FUNCTION_BLOCK FB_PostPalletizer EXTENDS FB_Chain
VAR_INPUT
END_VAR
VAR_OUTPUT
END_VAR
VAR
END_VAR

END_FUNCTION_BLOCK

(* stored: Version 1.1.0.1, ProductVersion 3.1.4024.0
   POU FB_PostPalletizer: Id {d145f42d-ec17-4f04-88d0-151eae25ee5d}, SpecialFunc None *)
